// TIA Portal V17 export
// export: Created 2024-09-02T12:50:33.7492909Z, ExportSetting WithDefaults, DisplayName Totally Integrated Automation Portal, DisplayVersion V17, DisplayName TIA Portal Openness, DisplayVersion V17, DisplayName TIA Portal Version Control Interface, DisplayVersion V17, DisplayName STEP 7 Professional, DisplayVersion V17, DisplayName STEP 7 Safety, DisplayVersion V17, DisplayName WinCC Professional, DisplayVersion V17
TYPE "TypeMobyAdressen"
TITLE = moby addresses / Mobyadressen
// stored: IsFailsafeCompliant false
   STRUCT
      OKfest { ExternalWritable := 'False'} : Bool;
      OKflex { ExternalWritable := 'False'} : Bool;
      FehlerEingabe { ExternalWritable := 'False'} : Bool;
      FehlerQdaten { ExternalWritable := 'False'} : Bool;
      Res4 { ExternalWritable := 'False'} : Bool;
      Res5 { ExternalWritable := 'False'} : Bool;
      Res6 { ExternalWritable := 'False'} : Bool;
      Res7 { ExternalWritable := 'False'} : Bool;
      PRG { ExternalWritable := 'False'} : DInt;
      KEY { ExternalWritable := 'False'} : DInt;
      TAF { ExternalWritable := 'False'} : DInt;
      DMC_SOLL { ExternalWritable := 'False'} : Array[1..8] of DInt;
      DMC_IST { ExternalWritable := 'False'} : Array[1..8] of DInt;
      DMC_IST_LN { ExternalWritable := 'False'} : Array[1..8] of DInt;
      MK_MIT { ExternalWritable := 'False'} : Array[1..8] of DInt;
      MK_OHNE { ExternalWritable := 'False'} : Array[1..8] of DInt;
      Q_DATEN_IST { ExternalWritable := 'False'} : DInt;
      Q_DATEN_IST_LN { ExternalWritable := 'False'} : DInt;
      PRG_VORSTAT : DInt;
   END_STRUCT;
END_TYPE
